KUKA KRL program: ps_603res_c1_orig.src, ps_603res_c1_orig.dat

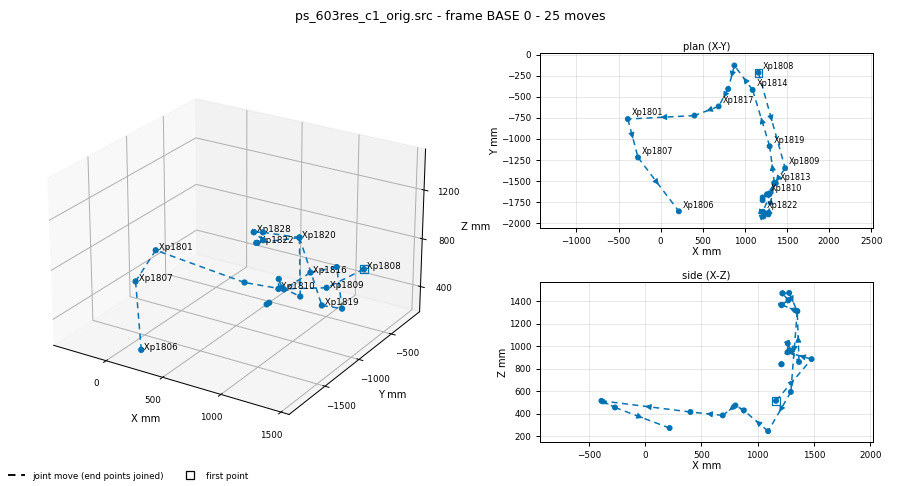
[picture p0: tool path of ps_603res_c1_orig.src in frame BASE 0, 25 of 40 moves have a stored position in this frame; points joined in program order, loops and branches not executed]
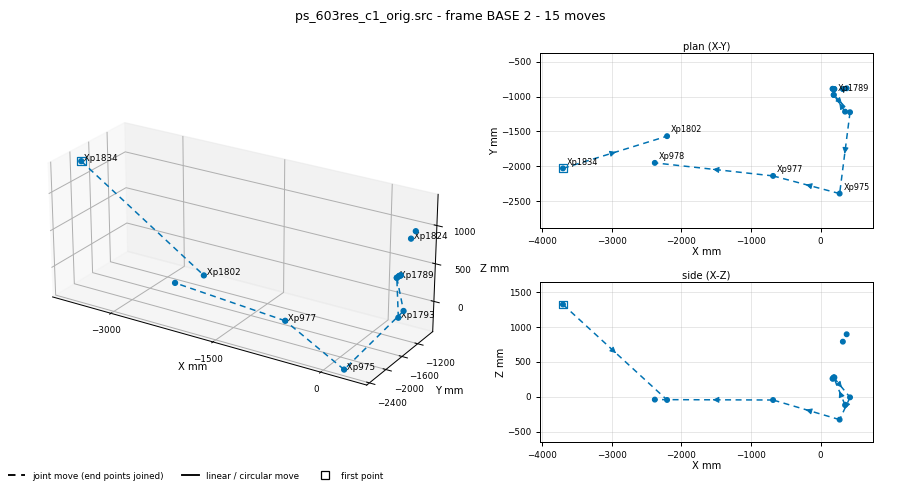
[picture p1: tool path of ps_603res_c1_orig.src in frame BASE 2, 15 of 40 moves have a stored position in this frame; points joined in program order, loops and branches not executed]
--- ps_603res_c1_orig.src ---
&ACCESS RVO
&COMMENT Solda Respot Geo1 C1
DEF ps_603res_c1_orig( )
EXT e_Fraes1 ( )
EXT f_Fraes1 ( )

  ;FOLD INI;%{PE}%V2.2.2,%MKUKATPBASIS,%CINIT,%VCOMMON,%P
  ;FOLD BAS INI;%{PE}%V2.2.2,%MKUKATPBASIS,%CINIT,%VINIT,%P
  INTERRUPT DECL 3 WHEN $STOPMESS==TRUE DO IR_STOPM ( )
  INTERRUPT ON 3
  BAS (#INITMOV,0 )
  ;ENDFOLD
  ;FOLD A20 INI;%{E}%V2.2.2,%MKUKATPA20,%CINIT,%VINIT,%P
  IF ARC20==TRUE THEN
    A20 (ARC_INI)
    INTERRUPT DECL 6 WHEN $CYCFLAG[3]==FALSE DO A20(TECH_STOP2)
  ENDIF
  ;ENDFOLD
  ;FOLD A10 INI;%{E}%V2.2.2,%MKUKATPARC,%CINIT,%VINIT,%P
  IF A10_OPTION==#ACTIVE THEN
    INTERRUPT DECL 4 WHEN $CYCFLAG[2]==FALSE DO A10 (#APPL_ERROR)
    INTERRUPT DECL 7 WHEN A_ARC_SWI==#ACTIVE DO A10 (#ARC_SEAM)
    INTERRUPT DECL 5 WHEN A_FLY_ARC==TRUE DO A10 (#HPU_ARC)
    INTERRUPT  ON 5
    A10_INI ( )
  ENDIF
  ;ENDFOLD
  ;FOLD GRIPPER INI;%{E}%V2.2.2,%MKUKATPGRIPPER,%CINIT,%VINIT,%P
  USER_GRP(0,DUMMY,DUMMY,GDEFAULT)
  ;ENDFOLD
  ;FOLD SPOT INI;%{E}%V.2.2,%MKUKATPSPOT,%CINIT,%VINIT,%P
  USERSPOT(#INIT)
  ;ENDFOLD
  ;FOLD TOUCHSENSE INI;%{E}%V2.2.2,%MKUKATPTS,%CINIT,%VINIT,%P
  IF H70_OPTION THEN
    INTERRUPT DECL 15 WHEN $MEAS_PULSE[TOUCH_I[TOUCH_ACTIVE].IN_NR] DO H70 (6,CD0 )
    INTERRUPT DECL 16 WHEN $ZERO_MOVE DO H70 (7,CD0 )
    INTERRUPT DECL 17 WHEN $TECHPAR_C[FG_TOUCH,8]>0.5 DO H70 (8,CD0)
    H70 (1,CD0 )
  ENDIF
  ;ENDFOLD
  ;FOLD USER INI;%{P}%V2.2.2,%MKUKATPUSER,%CINIT,%VINIT,%P
  ;Make your modifications here
  ;ENDFOLD
  ;ENDFOLD

; Caracterização dos meios de produção:
; Versão Atual:
; 19/07/2013 12:00 Name: P13.060-R3 CHANGES: Solda respot C1
; Accelo

chk_w1_wechs_ok ( )        ;VERIFICAÇÃO DE FERRAMENTA: C1

;FOLD PTP p1834  Vel= 80 % PDAT43 Tool[1]:Gun C1 Base[2]:Accelo;%{PE}%R 4.1.16,%MKUKATPBASIS,%CMOVE,%VPTP,%P 1:PTP, 2:p1834, 3:, 5:80, 7:PDAT43
$BWDSTART = FALSE
PDAT_ACT=PPDAT43
BAS(#PTP_DAT)
FDAT_ACT=Fp1834
BAS(#FRAMES)
BAS(#VEL_PTP,80)
PTP Xp1834
;ENDFOLD
;FOLD PTP p1802  Vel= 80 % PDAT11 Tool[1]:Gun C1 Base[2]:Accelo;%{PE}%R 4.1.16,%MKUKATPBASIS,%CMOVE,%VPTP,%P 1:PTP, 2:p1802, 3:, 5:80, 7:PDAT11
$BWDSTART = FALSE
PDAT_ACT=PPDAT11
BAS(#PTP_DAT)
FDAT_ACT=Fp1802
BAS(#FRAMES)
BAS(#VEL_PTP,80)
PTP Xp1802
;ENDFOLD

;FOLD OUT 838 'Solic. Lib. Soldar Respot GEO 1'  State= TRUE ;%{PE}%R 4.1.16,%MKUKATPBASIS,%COUT,%VOUTX,%P 2:838, 3:'Solic. Lib. Soldar Respot GEO 1', 5:TRUE, 6:
$OUT[838]=TRUE
;ENDFOLD
;FOLD WAIT FOR IN 846 'Aguarda lib. soldar respot Geo1'  State= TRUE ;%{PE}%R 4.1.16,%MKUKATPBASIS,%CWAIT_FOR,%VWAIT_FOR,%P 1:0, 2:846, 3:'Aguarda lib. soldar respot Geo1', 5:TRUE, 6:
WAIT FOR $IN[846]==TRUE
;ENDFOLD
;FOLD OUT 838 'Solic. Lib. Soldar Respot GEO 1'  State= FALSE ;%{PE}%R 4.1.16,%MKUKATPBASIS,%COUT,%VOUTX,%P 2:838, 3:'Solic. Lib. Soldar Respot GEO 1', 5:FALSE, 6:
$OUT[838]=FALSE
;ENDFOLD

;FOLD OUT 851 'Libera  AGV'  State= FALSE ;%{PE}%R 4.1.16,%MKUKATPBASIS,%COUT,%VOUTX,%P 2:851, 3:'Libera  AGV', 5:FALSE, 6:
$OUT[851]=FALSE
;ENDFOLD

;FOLD Kollision.Ueberwachung_1_Ein ;%{PE}%MKUKATPUSER
COLLSTOP( 1, 1 ) ;INTERRUPTUEBERWACHT
;ENDFOLD

;FOLD PTP p1808  Vel= 80 % PDAT17 Tool[1]:Gun C1 Base[0];%{PE}%R 4.1.16,%MKUKATPBASIS,%CMOVE,%VPTP,%P 1:PTP, 2:p1808, 3:, 5:80, 7:PDAT17
$BWDSTART = FALSE
PDAT_ACT=PPDAT17
BAS(#PTP_DAT)
FDAT_ACT=Fp1808
BAS(#FRAMES)
BAS(#VEL_PTP,80)
PTP Xp1808
;ENDFOLD
;FOLD PTP p1809 CONT Vel= 80 % PDAT18 Tool[1]:Gun C1 Base[0];%{PE}%R 4.1.16,%MKUKATPBASIS,%CMOVE,%VPTP,%P 1:PTP, 2:p1809, 3:C_PTP, 5:80, 7:PDAT18
$BWDSTART = FALSE
PDAT_ACT=PPDAT18
BAS(#PTP_DAT)
FDAT_ACT=Fp1809
BAS(#FRAMES)
BAS(#VEL_PTP,80)
PTP Xp1809 C_PTP
;ENDFOLD
;FOLD PTP p1810 CONT Vel= 80 % PDAT19 Tool[1]:Gun C1 Base[0];%{PE}%R 4.1.16,%MKUKATPBASIS,%CMOVE,%VPTP,%P 1:PTP, 2:p1810, 3:C_PTP, 5:80, 7:PDAT19
$BWDSTART = FALSE
PDAT_ACT=PPDAT19
BAS(#PTP_DAT)
FDAT_ACT=Fp1810
BAS(#FRAMES)
BAS(#VEL_PTP,80)
PTP Xp1810 C_PTP
;ENDFOLD

;FOLD PTP SWP_62_0005 PDAT20 SPOT Gun= 1 RETR OPN PgNo1= 36 ACTIVE= 1 Tool[1]:Gun C1 Base[0];%{PE}%R 4.1.12,%MKUKATPSPOT,%CSPOT,%VPTP,%P 1:PTP, 2:SWP_62_0005, 3:, 5:80, 7:PDAT20, 10:1, 12:#FIRST, 14:#OPN, 16:36, 18:1, 20:0, 22:0, 24:1, 25:NORMAL
$BWDSTART = FALSE
PDAT_ACT=PPDAT20
BAS(#PTP_DAT)
FDAT_ACT=FSWP_62_0005
BAS(#FRAMES)
BAS(#VEL_PTP,PPDAT20.VEL)
S_ACT.GUN=1
S_ACT.PAIR=SDEFAULT.PAIR
S_ACT.RETR=#OPN
S_ACT.CLO_TM=1
S_ACT.PGNO1=36
S_ACT.PGNO2=SDEFAULT.PGNO2
S_ACT.PRESS1=SDEFAULT.PRESS1
S_ACT.PRESS2=SDEFAULT.PRESS2
S_READY=FALSE
PTP XSWP_62_0005
USERSPOT(#SPOT, S_ACT)
WAIT FOR S_READY
;ENDFOLD

;FOLD PTP p1812 CONT Vel= 80 % PDAT21 Tool[1]:Gun C1 Base[0];%{PE}%R 4.1.16,%MKUKATPBASIS,%CMOVE,%VPTP,%P 1:PTP, 2:p1812, 3:C_PTP, 5:80, 7:PDAT21
$BWDSTART = FALSE
PDAT_ACT=PPDAT21
BAS(#PTP_DAT)
FDAT_ACT=Fp1812
BAS(#FRAMES)
BAS(#VEL_PTP,80)
PTP Xp1812 C_PTP
;ENDFOLD
;FOLD PTP p1813 CONT Vel= 80 % PDAT22 Tool[1]:Gun C1 Base[0];%{PE}%R 4.1.16,%MKUKATPBASIS,%CMOVE,%VPTP,%P 1:PTP, 2:p1813, 3:C_PTP, 5:80, 7:PDAT22
$BWDSTART = FALSE
PDAT_ACT=PPDAT22
BAS(#PTP_DAT)
FDAT_ACT=Fp1813
BAS(#FRAMES)
BAS(#VEL_PTP,80)
PTP Xp1813 C_PTP
;ENDFOLD
;FOLD PTP p1820  Vel= 80 % PDAT29 Tool[1]:Gun C1 Base[0];%{PE}%R 4.1.16,%MKUKATPBASIS,%CMOVE,%VPTP,%P 1:PTP, 2:p1820, 3:, 5:80, 7:PDAT29
$BWDSTART = FALSE
PDAT_ACT=PPDAT29
BAS(#PTP_DAT)
FDAT_ACT=Fp1820
BAS(#FRAMES)
BAS(#VEL_PTP,80)
PTP Xp1820
;ENDFOLD
;FOLD PTP p1822  Vel= 80 % PDAT31 Tool[1]:Gun C1 Base[0];%{PE}%R 4.1.16,%MKUKATPBASIS,%CMOVE,%VPTP,%P 1:PTP, 2:p1822, 3:, 5:80, 7:PDAT31
$BWDSTART = FALSE
PDAT_ACT=PPDAT31
BAS(#PTP_DAT)
FDAT_ACT=Fp1822
BAS(#FRAMES)
BAS(#VEL_PTP,80)
PTP Xp1822
;ENDFOLD

;FOLD PTP p1824 PDAT33 SPOT Gun= 1 RETR OPN PgNo1= 1 ACTIVE= 1 Tool[1]:Gun C1 Base[2]:Accelo;%{PE}%R 4.1.12,%MKUKATPSPOT,%CSPOT,%VPTP,%P 1:PTP, 2:p1824, 3:, 5:80, 7:PDAT33, 10:1, 12:#FIRST, 14:#OPN, 16:1, 18:1, 20:0, 22:0, 24:1, 25:NORMAL
$BWDSTART = FALSE
PDAT_ACT=PPDAT33
BAS(#PTP_DAT)
FDAT_ACT=Fp1824
BAS(#FRAMES)
BAS(#VEL_PTP,PPDAT33.VEL)
S_ACT.GUN=1
S_ACT.PAIR=SDEFAULT.PAIR
S_ACT.RETR=#OPN
S_ACT.CLO_TM=1
S_ACT.PGNO1=1
S_ACT.PGNO2=SDEFAULT.PGNO2
S_ACT.PRESS1=SDEFAULT.PRESS1
S_ACT.PRESS2=SDEFAULT.PRESS2
S_READY=FALSE
PTP Xp1824
USERSPOT(#SPOT, S_ACT)
WAIT FOR S_READY
;ENDFOLD

;FOLD PTP p1825  Vel= 80 % PDAT34 Tool[1]:Gun C1 Base[0];%{PE}%R 4.1.16,%MKUKATPBASIS,%CMOVE,%VPTP,%P 1:PTP, 2:p1825, 3:, 5:80, 7:PDAT34
$BWDSTART = FALSE
PDAT_ACT=PPDAT34
BAS(#PTP_DAT)
FDAT_ACT=Fp1825
BAS(#FRAMES)
BAS(#VEL_PTP,80)
PTP Xp1825
;ENDFOLD
;FOLD PTP p1826  Vel= 80 % PDAT35 Tool[1]:Gun C1 Base[0];%{PE}%R 4.1.16,%MKUKATPBASIS,%CMOVE,%VPTP,%P 1:PTP, 2:p1826, 3:, 5:80, 7:PDAT35
$BWDSTART = FALSE
PDAT_ACT=PPDAT35
BAS(#PTP_DAT)
FDAT_ACT=Fp1826
BAS(#FRAMES)
BAS(#VEL_PTP,80)
PTP Xp1826
;ENDFOLD
;FOLD PTP p1828  Vel= 80 % PDAT37 Tool[1]:Gun C1 Base[0];%{PE}%R 4.1.16,%MKUKATPBASIS,%CMOVE,%VPTP,%P 1:PTP, 2:p1828, 3:, 5:80, 7:PDAT37
$BWDSTART = FALSE
PDAT_ACT=PPDAT37
BAS(#PTP_DAT)
FDAT_ACT=Fp1828
BAS(#FRAMES)
BAS(#VEL_PTP,80)
PTP Xp1828
;ENDFOLD

;FOLD PTP p1829 PDAT38 SPOT Gun= 1 RETR OPN PgNo1= 1 ACTIVE= 1 Tool[1]:Gun C1 Base[2]:Accelo;%{PE}%R 4.1.12,%MKUKATPSPOT,%CSPOT,%VPTP,%P 1:PTP, 2:p1829, 3:, 5:80, 7:PDAT38, 10:1, 12:#FIRST, 14:#OPN, 16:1, 18:1, 20:0, 22:0, 24:1, 25:NORMAL
$BWDSTART = FALSE
PDAT_ACT=PPDAT38
BAS(#PTP_DAT)
FDAT_ACT=Fp1829
BAS(#FRAMES)
BAS(#VEL_PTP,PPDAT38.VEL)
S_ACT.GUN=1
S_ACT.PAIR=SDEFAULT.PAIR
S_ACT.RETR=#OPN
S_ACT.CLO_TM=1
S_ACT.PGNO1=1
S_ACT.PGNO2=SDEFAULT.PGNO2
S_ACT.PRESS1=SDEFAULT.PRESS1
S_ACT.PRESS2=SDEFAULT.PRESS2
S_READY=FALSE
PTP Xp1829
USERSPOT(#SPOT, S_ACT)
WAIT FOR S_READY
;ENDFOLD

;FOLD PTP p1830  Vel= 80 % PDAT39 Tool[1]:Gun C1 Base[0];%{PE}%R 4.1.16,%MKUKATPBASIS,%CMOVE,%VPTP,%P 1:PTP, 2:p1830, 3:, 5:80, 7:PDAT39
$BWDSTART = FALSE
PDAT_ACT=PPDAT39
BAS(#PTP_DAT)
FDAT_ACT=Fp1830
BAS(#FRAMES)
BAS(#VEL_PTP,80)
PTP Xp1830
;ENDFOLD
;FOLD PTP p1831  Vel= 80 % PDAT40 Tool[1]:Gun C1 Base[0];%{PE}%R 4.1.16,%MKUKATPBASIS,%CMOVE,%VPTP,%P 1:PTP, 2:p1831, 3:, 5:80, 7:PDAT40
$BWDSTART = FALSE
PDAT_ACT=PPDAT40
BAS(#PTP_DAT)
FDAT_ACT=Fp1831
BAS(#FRAMES)
BAS(#VEL_PTP,80)
PTP Xp1831
;ENDFOLD
;FOLD PTP p1832  Vel= 80 % PDAT41 Tool[1]:Gun C1 Base[0];%{PE}%R 4.1.16,%MKUKATPBASIS,%CMOVE,%VPTP,%P 1:PTP, 2:p1832, 3:, 5:80, 7:PDAT41
$BWDSTART = FALSE
PDAT_ACT=PPDAT41
BAS(#PTP_DAT)
FDAT_ACT=Fp1832
BAS(#FRAMES)
BAS(#VEL_PTP,80)
PTP Xp1832
;ENDFOLD
;FOLD PTP p1819  Vel= 80 % PDAT28 Tool[1]:Gun C1 Base[0];%{PE}%R 4.1.16,%MKUKATPBASIS,%CMOVE,%VPTP,%P 1:PTP, 2:p1819, 3:, 5:80, 7:PDAT28
$BWDSTART = FALSE
PDAT_ACT=PPDAT28
BAS(#PTP_DAT)
FDAT_ACT=Fp1819
BAS(#FRAMES)
BAS(#VEL_PTP,80)
PTP Xp1819
;ENDFOLD
;FOLD PTP p1814 CONT Vel= 80 % PDAT23 Tool[1]:Gun C1 Base[0];%{PE}%R 4.1.16,%MKUKATPBASIS,%CMOVE,%VPTP,%P 1:PTP, 2:p1814, 3:C_PTP, 5:80, 7:PDAT23
$BWDSTART = FALSE
PDAT_ACT=PPDAT23
BAS(#PTP_DAT)
FDAT_ACT=Fp1814
BAS(#FRAMES)
BAS(#VEL_PTP,80)
PTP Xp1814 C_PTP
;ENDFOLD
;FOLD PTP p1815 CONT Vel= 80 % PDAT24 Tool[1]:Gun C1 Base[0];%{PE}%R 4.1.16,%MKUKATPBASIS,%CMOVE,%VPTP,%P 1:PTP, 2:p1815, 3:C_PTP, 5:80, 7:PDAT24
$BWDSTART = FALSE
PDAT_ACT=PPDAT24
BAS(#PTP_DAT)
FDAT_ACT=Fp1815
BAS(#FRAMES)
BAS(#VEL_PTP,80)
PTP Xp1815 C_PTP
;ENDFOLD
;FOLD PTP p1816 CONT Vel= 80 % PDAT25 Tool[1]:Gun C1 Base[0];%{PE}%R 4.1.16,%MKUKATPBASIS,%CMOVE,%VPTP,%P 1:PTP, 2:p1816, 3:C_PTP, 5:80, 7:PDAT25
$BWDSTART = FALSE
PDAT_ACT=PPDAT25
BAS(#PTP_DAT)
FDAT_ACT=Fp1816
BAS(#FRAMES)
BAS(#VEL_PTP,80)
PTP Xp1816 C_PTP
;ENDFOLD
;FOLD PTP p1817 CONT Vel= 80 % PDAT26 Tool[1]:Gun C1 Base[0];%{PE}%R 4.1.16,%MKUKATPBASIS,%CMOVE,%VPTP,%P 1:PTP, 2:p1817, 3:C_PTP, 5:80, 7:PDAT26
$BWDSTART = FALSE
PDAT_ACT=PPDAT26
BAS(#PTP_DAT)
FDAT_ACT=Fp1817
BAS(#FRAMES)
BAS(#VEL_PTP,80)
PTP Xp1817 C_PTP
;ENDFOLD
;FOLD PTP p1818 CONT Vel= 80 % PDAT27 Tool[1]:Gun C1 Base[0];%{PE}%R 4.1.16,%MKUKATPBASIS,%CMOVE,%VPTP,%P 1:PTP, 2:p1818, 3:C_PTP, 5:80, 7:PDAT27
$BWDSTART = FALSE
PDAT_ACT=PPDAT27
BAS(#PTP_DAT)
FDAT_ACT=Fp1818
BAS(#FRAMES)
BAS(#VEL_PTP,80)
PTP Xp1818 C_PTP
;ENDFOLD
;FOLD PTP p1801 CONT Vel= 80 % PDAT10 Tool[1]:Gun C1 Base[0];%{PE}%R 4.1.16,%MKUKATPBASIS,%CMOVE,%VPTP,%P 1:PTP, 2:p1801, 3:C_PTP, 5:80, 7:PDAT10
$BWDSTART = FALSE
PDAT_ACT=PPDAT10
BAS(#PTP_DAT)
FDAT_ACT=Fp1801
BAS(#FRAMES)
BAS(#VEL_PTP,80)
PTP Xp1801 C_PTP
;ENDFOLD
;FOLD PTP p1807 CONT Vel= 80 % PDAT16 Tool[1]:Gun C1 Base[0];%{PE}%R 4.1.16,%MKUKATPBASIS,%CMOVE,%VPTP,%P 1:PTP, 2:p1807, 3:C_PTP, 5:80, 7:PDAT16
$BWDSTART = FALSE
PDAT_ACT=PPDAT16
BAS(#PTP_DAT)
FDAT_ACT=Fp1807
BAS(#FRAMES)
BAS(#VEL_PTP,80)
PTP Xp1807 C_PTP
;ENDFOLD
;FOLD PTP p1806  Vel= 80 % PDAT15 Tool[1]:Gun C1 Base[0];%{PE}%R 4.1.16,%MKUKATPBASIS,%CMOVE,%VPTP,%P 1:PTP, 2:p1806, 3:, 5:80, 7:PDAT15
$BWDSTART = FALSE
PDAT_ACT=PPDAT15
BAS(#PTP_DAT)
FDAT_ACT=Fp1806
BAS(#FRAMES)
BAS(#VEL_PTP,80)
PTP Xp1806
;ENDFOLD

;FOLD OUT 838 'Solic. Lib. Soldar Respot GEO 1'  State= TRUE ;%{PE}%R 4.1.16,%MKUKATPBASIS,%COUT,%VOUTX,%P 2:838, 3:'Solic. Lib. Soldar Respot GEO 1', 5:TRUE, 6:
$OUT[838]=TRUE
;ENDFOLD
;FOLD WAIT FOR IN 846 'aguarda lib. soldar respot Geo1'  State= TRUE ;%{PE}%R 4.1.16,%MKUKATPBASIS,%CWAIT_FOR,%VWAIT_FOR,%P 1:0, 2:846, 3:'aguarda lib. soldar respot Geo1', 5:TRUE, 6:
WAIT FOR $IN[846]==TRUE
;ENDFOLD
;FOLD OUT 838 'Solic. Lib. Soldar Respot GEO 1'  State= FALSE ;%{PE}%R 4.1.16,%MKUKATPBASIS,%COUT,%VOUTX,%P 2:838, 3:'Solic. Lib. Soldar Respot GEO 1', 5:FALSE, 6:
$OUT[838]=FALSE
;ENDFOLD

;FOLD PTP p1793 CONT Vel= 65 % PDAT7 Tool[1]:Gun C1 Base[2]:Accelo;%{PE}%R 4.1.16,%MKUKATPBASIS,%CMOVE,%VPTP,%P 1:PTP, 2:p1793, 3:C_PTP, 5:65, 7:PDAT7
$BWDSTART = FALSE
PDAT_ACT=PPDAT7
BAS(#PTP_DAT)
FDAT_ACT=Fp1793
BAS(#FRAMES)
BAS(#VEL_PTP,65)
PTP Xp1793 C_PTP
;ENDFOLD
;FOLD PTP p1789  Vel= 75 % PDAT3 Tool[1]:Gun C1 Base[2]:Accelo;%{PE}%R 4.1.16,%MKUKATPBASIS,%CMOVE,%VPTP,%P 1:PTP, 2:p1789, 3:, 5:75, 7:PDAT3
$BWDSTART = FALSE
PDAT_ACT=PPDAT3
BAS(#PTP_DAT)
FDAT_ACT=Fp1789
BAS(#FRAMES)
BAS(#VEL_PTP,75)
PTP Xp1789
;ENDFOLD

;FOLD OUT 839 'Soldando'  State= TRUE ;%{PE}%R 4.1.16,%MKUKATPBASIS,%COUT,%VOUTX,%P 2:839, 3:'Soldando', 5:TRUE, 6:
$OUT[839]=TRUE
;ENDFOLD
;FOLD OUT 848 'Area de Solda'  State= FALSE ;%{PE}%R 4.1.16,%MKUKATPBASIS,%COUT,%VOUTX,%P 2:848, 3:'Area de Solda', 5:FALSE, 6:
$OUT[848]=FALSE
;ENDFOLD

;FOLD LIN p1794 CONT Vel= 2 m/s CPDAT14 Tool[1]:Gun C1 Base[2]:Accelo;%{PE}%R 4.1.16,%MKUKATPBASIS,%CMOVE,%VLIN,%P 1:LIN, 2:p1794, 3:C_DIS, 5:2, 7:CPDAT14
$BWDSTART = FALSE
LDAT_ACT=LCPDAT14
BAS(#CP_DAT)
FDAT_ACT=Fp1794
BAS(#FRAMES)
BAS(#VEL_CP,2)
LIN Xp1794 C_DIS
;ENDFOLD

;FOLD ; SWP_60_0213;%{PE}%R 4.1.16,%MKUKATPBASIS,%CCOMMENT,%VNORMAL,%P 2:SWP_60_0213
;ENDFOLD
;FOLD LIN swp_60_0213 CPDAT16 SPOT Gun= 1 RETR OPN PgNo1= 14 ACTIVE= 1 Tool[1]:Gun C1 Base[0];%{PE}%R 4.1.12,%MKUKATPSPOT,%CSPOT,%VLIN,%P 1:LIN, 2:swp_60_0213, 3:, 5:2, 7:CPDAT16, 10:1, 12:#FIRST, 14:#OPN, 16:14, 18:1, 20:0, 22:0, 24:1, 25:NORMAL
$BWDSTART = FALSE
LDAT_ACT=LCPDAT16
BAS(#CP_DAT)
FDAT_ACT=Fswp_60_0213
BAS(#FRAMES)
BAS(#VEL_CP,LCPDAT16.VEL)
S_ACT.GUN=1
S_ACT.PAIR=SDEFAULT.PAIR
S_ACT.RETR=#OPN
S_ACT.CLO_TM=1
S_ACT.PGNO1=14
S_ACT.PGNO2=SDEFAULT.PGNO2
S_ACT.PRESS1=SDEFAULT.PRESS1
S_ACT.PRESS2=SDEFAULT.PRESS2
S_READY=FALSE
LIN Xswp_60_0213
USERSPOT(#SPOT, S_ACT)
WAIT FOR S_READY
;ENDFOLD

;FOLD LIN p1795 CONT Vel= 2 m/s CPDAT15 Tool[1]:Gun C1 Base[2]:Accelo;%{PE}%R 4.1.16,%MKUKATPBASIS,%CMOVE,%VLIN,%P 1:LIN, 2:p1795, 3:C_DIS, 5:2, 7:CPDAT15
$BWDSTART = FALSE
LDAT_ACT=LCPDAT15
BAS(#CP_DAT)
FDAT_ACT=Fp1795
BAS(#FRAMES)
BAS(#VEL_CP,2)
LIN Xp1795 C_DIS
;ENDFOLD

;FOLD ; SWP_60_0215;%{PE}%R 4.1.16,%MKUKATPBASIS,%CCOMMENT,%VNORMAL,%P 2:SWP_60_0215
;ENDFOLD
;FOLD LIN swp_60_0215 CPDAT19 SPOT Gun= 1 RETR OPN PgNo1= 15 ACTIVE= 1 Tool[1]:Gun C1 Base[0];%{PE}%R 4.1.12,%MKUKATPSPOT,%CSPOT,%VLIN,%P 1:LIN, 2:swp_60_0215, 3:, 5:2, 7:CPDAT19, 10:1, 12:#FIRST, 14:#OPN, 16:15, 18:1, 20:0, 22:0, 24:1, 25:NORMAL
$BWDSTART = FALSE
LDAT_ACT=LCPDAT19
BAS(#CP_DAT)
FDAT_ACT=Fswp_60_0215
BAS(#FRAMES)
BAS(#VEL_CP,LCPDAT19.VEL)
S_ACT.GUN=1
S_ACT.PAIR=SDEFAULT.PAIR
S_ACT.RETR=#OPN
S_ACT.CLO_TM=1
S_ACT.PGNO1=15
S_ACT.PGNO2=SDEFAULT.PGNO2
S_ACT.PRESS1=SDEFAULT.PRESS1
S_ACT.PRESS2=SDEFAULT.PRESS2
S_READY=FALSE
LIN Xswp_60_0215
USERSPOT(#SPOT, S_ACT)
WAIT FOR S_READY
;ENDFOLD

;FOLD LIN p1797 CONT Vel= 2 m/s CPDAT18 Tool[1]:Gun C1 Base[2]:Accelo;%{PE}%R 4.1.16,%MKUKATPBASIS,%CMOVE,%VLIN,%P 1:LIN, 2:p1797, 3:C_DIS, 5:2, 7:CPDAT18
$BWDSTART = FALSE
LDAT_ACT=LCPDAT18
BAS(#CP_DAT)
FDAT_ACT=Fp1797
BAS(#FRAMES)
BAS(#VEL_CP,2)
LIN Xp1797 C_DIS
;ENDFOLD

;FOLD OUT 839 'Soldando'  State= FALSE ;%{PE}%R 4.1.16,%MKUKATPBASIS,%COUT,%VOUTX,%P 2:839, 3:'Soldando', 5:FALSE, 6:
$OUT[839]=FALSE
;ENDFOLD
;FOLD OUT 848 'Area de Solda'  State= TRUE ;%{PE}%R 4.1.16,%MKUKATPBASIS,%COUT,%VOUTX,%P 2:848, 3:'Area de Solda', 5:TRUE, 6:
$OUT[848]=TRUE
;ENDFOLD

;FOLD LIN p1798 CONT Vel= 2 m/s CPDAT20 Tool[1]:Gun C1 Base[2]:Accelo;%{PE}%R 4.1.16,%MKUKATPBASIS,%CMOVE,%VLIN,%P 1:LIN, 2:p1798, 3:C_DIS, 5:2, 7:CPDAT20
$BWDSTART = FALSE
LDAT_ACT=LCPDAT20
BAS(#CP_DAT)
FDAT_ACT=Fp1798
BAS(#FRAMES)
BAS(#VEL_CP,2)
LIN Xp1798 C_DIS
;ENDFOLD

;FOLD PTP p973 CONT Vel= 80 % P_OLP11 Tool[1]:Gun C1 Base[2]:Accelo;%{PE}%R 4.1.16,%MKUKATPBASIS,%CMOVE,%VPTP,%P 1:PTP, 2:p973, 3:C_PTP, 5:80, 7:P_OLP11
$BWDSTART = FALSE
PDAT_ACT=PP_OLP11
BAS(#PTP_DAT)
FDAT_ACT=Fp973
BAS(#FRAMES)
BAS(#VEL_PTP,80)
PTP Xp973 C_PTP
;ENDFOLD
;FOLD PTP p974 CONT Vel= 80 % P_OLP12 Tool[1]:Gun C1 Base[2]:Accelo;%{PE}%R 4.1.16,%MKUKATPBASIS,%CMOVE,%VPTP,%P 1:PTP, 2:p974, 3:C_PTP, 5:80, 7:P_OLP12
$BWDSTART = FALSE
PDAT_ACT=PP_OLP12
BAS(#PTP_DAT)
FDAT_ACT=Fp974
BAS(#FRAMES)
BAS(#VEL_PTP,80)
PTP Xp974 C_PTP
;ENDFOLD
;FOLD PTP p975 CONT Vel= 80 % P_OLP13 Tool[1]:Gun C1 Base[2]:Accelo;%{PE}%R 4.1.16,%MKUKATPBASIS,%CMOVE,%VPTP,%P 1:PTP, 2:p975, 3:C_PTP, 5:80, 7:P_OLP13
$BWDSTART = FALSE
PDAT_ACT=PP_OLP13
BAS(#PTP_DAT)
FDAT_ACT=Fp975
BAS(#FRAMES)
BAS(#VEL_PTP,80)
PTP Xp975 C_PTP
;ENDFOLD
;FOLD PTP p977  Vel= 80 % P_OLP15 Tool[1]:Gun C1 Base[2]:Accelo;%{PE}%R 4.1.16,%MKUKATPBASIS,%CMOVE,%VPTP,%P 1:PTP, 2:p977, 3:, 5:80, 7:P_OLP15
$BWDSTART = FALSE
PDAT_ACT=PP_OLP15
BAS(#PTP_DAT)
FDAT_ACT=Fp977
BAS(#FRAMES)
BAS(#VEL_PTP,80)
PTP Xp977
;ENDFOLD

;FOLD ; END INTERLOCK COM R1;%{PE}%R 4.1.16,%MKUKATPBASIS,%CCOMMENT,%VNORMAL,%P 2:END INTERLOCK COM R1
;ENDFOLD
;FOLD Kollision.Ueberwachung_1_Aus ;%{PE}%MKUKATPUSER
COLLSTOP( 1, 2 )
;ENDFOLD

;FOLD PULSE 846 'R3 solda respot Geo 1 concluida'  State= TRUE   Time= 3 sec;%{PE}%R 4.1.16,%MKUKATPBASIS,%COUT,%VPULSE,%P 2:846, 3:'R3 solda respot Geo 1 concluida', 5:TRUE, 6:, 8:3
PULSE($OUT[846], TRUE,3)
;ENDFOLD

;FOLD PTP p978 CONT Vel= 100 % P_OLP16 Tool[1]:Gun C1 Base[2]:Accelo;%{PE}%R 4.1.16,%MKUKATPBASIS,%CMOVE,%VPTP,%P 1:PTP, 2:p978, 3:C_PTP, 5:100, 7:P_OLP16
$BWDSTART = FALSE
PDAT_ACT=PP_OLP16
BAS(#PTP_DAT)
FDAT_ACT=Fp978
BAS(#FRAMES)
BAS(#VEL_PTP,100)
PTP Xp978 C_PTP
;ENDFOLD

IF ((GHOST() OR $IN[821])) THEN
;FOLD OUT 176 'Proteção da pinca 2 fechar'  State= FALSE ;%{PE}%R 4.1.16,%MKUKATPBASIS,%COUT,%VOUTX,%P 2:176, 3:'Proteção da pinca 2 fechar', 5:FALSE, 6:
$OUT[176]=FALSE
;ENDFOLD
;FOLD OUT 175 'Proteção da pinca 2 abrir'  State= TRUE ;%{PE}%R 4.1.16,%MKUKATPBASIS,%COUT,%VOUTX,%P 2:175, 3:'Proteção da pinca 2 abrir', 5:TRUE, 6:
$OUT[175]=TRUE
;ENDFOLD
ENDIF

END

--- ps_603res_c1_orig.dat ---
&ACCESS RVO
&COMMENT Solda Respot Geo1 C1
DEFDAT ps_603res_c1_orig
;FOLD EXTERNAL DECLARATIONS;%{PE}%V2.2.2,%MKUKATPBASIS,%CEXT,%VCOMMON,%P
;FOLD BAS EXT;%{PE}%V2.2.2,%MKUKATPBASIS,%CEXT,%VEXT,%P
EXT  BAS (BAS_COMMAND  :IN,REAL  :IN )
DECL INT SUCCESS
;ENDFOLD
;FOLD A10 EXT;%{E}%V2.2.2,%MKUKATPARC,%CEXT,%VEXT,%P
EXT  A10 (A_CMD_T  :IN,A_STRT_T  :IN,A_WELD_T  :IN,A_END_T  :IN,INT  :IN )
;ENDFOLD
;FOLD A20 EXT;%{E}%V2.2.2,%MKUKATPA20,%CEXT,%VEXT,%P
EXT  A20 (INT  :IN,WELD_ST  :IN,WELD_FI  :IN,INT  :IN )
;ENDFOLD
;FOLD GRIPPER EXT;%{E}%V2.2.2,%MKUKATPGRIPPER,%CEXT,%VEXT,%P
EXT  H50 (INT  :IN,INT  :IN,INT  :IN,GRP_TYP  :IN )
;ENDFOLD
;FOLD SPOT EXT;%{E}%V2.2.2,%MKUKATPSPOT,%CEXT,%VEXT,%P
EXT  USERSPOT (S_COMMAND  :IN,SPOT_TYPE  :IN )
;ENDFOLD
;FOLD TOUCHSENSE EXT;%{E}%V2.2.2,%MKUKATPTS,%CEXT,%VEXT,%P
EXT  H70 (INT  :IN,SRCH_TYP_2  :OUT,E6POS  :IN,SRCH_TYP_3  :IN,SRCH_TYP_2  :IN,SRCH_TYP_2  :IN,SRCH_TYP_2  :IN,SRCH_TYP_2  :IN,SRCH_TYP_2  :IN,INT  :IN )
;ENDFOLD
;FOLD USER EXT;%{}%V2.2.2,%MKUKATPUSER,%CEXT,%VEXT,%P
;Make here your modifications
;ENDFOLD
;ENDFOLD

;# ============ START PATH : swp_p13060r3_ltc_resp1_c1 =============
DECL FDAT Fp963={TOOL_NO 1,BASE_NO 2,IPO_FRAME #BASE}
DECL PDAT PP_OLP1={VEL 100.0,ACC 100.0,APO_DIST 0.0}
DECL E6POS Xp963={x -3572.9751,y -2107.74902,z 1272.901,a 86.0327988,b 14.4777002,c 74.495903,s 2,t 3}
DECL FDAT Fp964={TOOL_NO 1,BASE_NO 2,IPO_FRAME #BASE}
DECL PDAT PP_OLP2={VEL 100.0,ACC 85.0,APO_DIST 60.0}
DECL E6POS Xp964={x -1796.38599,y -2237.50098,z 3255.19995,a -90.0,b 0.0,c 170.0,s 6,t 51}
DECL FDAT Fp965={TOOL_NO 1,BASE_NO 2,IPO_FRAME #BASE}
DECL PDAT PP_OLP3={VEL 100.0,ACC 85.0,APO_DIST 15.0}
DECL E6POS Xp965={x -1013.56299,y -2243.53296,z 3255.19995,a 70.0,b 0.0,c 170.0,s 6,t 50}
DECL FDAT Fp966={TOOL_NO 1,BASE_NO 2,IPO_FRAME #BASE}
DECL PDAT PP_OLP4={VEL 100.0,ACC 85.0,APO_DIST 20.0}
DECL E6POS Xp966={x -134.343201,y -2313.625,z -64.5488205,a 1.681077,b -1.44535995,c 0.678022921,s 2,t 10,e1 0.0,e2 0.0,e3 0.0,e4 0.0,e5 0.0,e6 0.0}
DECL FDAT Fp967={TOOL_NO 1,BASE_NO 2,IPO_FRAME #BASE}
DECL PDAT PP_OLP5={VEL 100.0,ACC 100.0,APO_DIST 100.0}
DECL E6POS Xp967={x 199.132004,y -934.976013,z 255.951996,a 31.1662006,b 48.9373016,c 116.802299,s 6,t 50}
DECL FDAT Fp968={TOOL_NO 1,BASE_NO 2,IPO_FRAME #BASE}
DECL PDAT PP_OLP6={VEL 100.0,ACC 85.0,APO_DIST 10.0}
DECL E6POS Xp968={x 318.066895,y -1890.32605,z -296.505615,a 6.09352779,b -3.63016009,c 11.6354103,s 2,t 10,e1 0.0,e2 0.0,e3 0.0,e4 0.0,e5 0.0,e6 0.0}
DECL FDAT Fp969={TOOL_NO 1,BASE_NO 2,IPO_FRAME #BASE}
DECL PDAT PP_OLP7={VEL 100.0,ACC 85.0,APO_DIST 5.0}
DECL E6POS Xp969={x 197.508408,y -888.166077,z 282.583313,a 2.79331207,b 35.6193008,c 91.0491791,s 6,t 50,e1 0.0,e2 0.0,e3 0.0,e4 0.0,e5 0.0,e6 0.0}
DECL FDAT Fp970={TOOL_NO 1,BASE_NO 2,IPO_FRAME #BASE}
DECL PDAT PP_OLP8={VEL 100.0,ACC 100.0,APO_DIST 100.0}
DECL E6POS Xp970={x 191.053497,y -889.268982,z 200.622604,a 2.60313106,b 52.9382095,c 92.072197,s 6,t 50,e1 0.0,e2 0.0,e3 0.0,e4 0.0,e5 0.0,e6 0.0}
DECL FDAT Fp971={TOOL_NO 1,BASE_NO 2,IPO_FRAME #BASE}
DECL PDAT PP_OLP9={VEL 100.0,ACC 100.0,APO_DIST 100.0}
DECL E6POS Xp971={x 193.593796,y -886.93158,z 200.001999,a 2.60292602,b 52.9385605,c 92.071907,s 6,t 50,e1 0.0,e2 0.0,e3 0.0,e4 0.0,e5 0.0,e6 0.0}
DECL FDAT Fp972={TOOL_NO 1,BASE_NO 2,IPO_FRAME #BASE}
DECL PDAT PP_OLP10={VEL 100.0,ACC 100.0,APO_DIST 100.0}
DECL E6POS Xp972={x 190.962006,y -887.40802,z 255.615005,a 15.6997004,b 59.0479012,c 103.552902,s 6,t 50}
DECL FDAT Fp973={TOOL_NO 1,BASE_NO 2,IPO_FRAME #BASE}
DECL PDAT PP_OLP11={VEL 100.0,ACC 85.0,APO_DIST 15.0}
DECL E6POS Xp973={x 188.3909,y -976.163513,z 275.360504,a 6.09893894,b 13.9292002,c 94.6382599,s 2,t 10,e1 0.0,e2 0.0,e3 0.0,e4 0.0,e5 0.0,e6 0.0}
DECL FDAT Fp974={TOOL_NO 1,BASE_NO 2,IPO_FRAME #BASE}
DECL PDAT PP_OLP12={VEL 100.0,ACC 85.0,APO_DIST 5.0}
DECL E6POS Xp974={x 422.566498,y -1224.58105,z -8.89597225,a 3.03044891,b -9.06613731,c 48.4070282,s 2,t 10,e1 0.0,e2 0.0,e3 0.0,e4 0.0,e5 0.0,e6 0.0}
DECL FDAT Fp975={TOOL_NO 1,BASE_NO 2,IPO_FRAME #BASE}
DECL PDAT PP_OLP13={VEL 100.0,ACC 85.0,APO_DIST 50.0}
DECL E6POS Xp975={x 273.068604,y -2393.427,z -329.290314,a 5.52923822,b -0.604498804,c -3.24042201,s 2,t 2,e1 0.0,e2 0.0,e3 0.0,e4 0.0,e5 0.0,e6 0.0}
DECL FDAT Fp976={TOOL_NO 1,BASE_NO 2,IPO_FRAME #BASE}
DECL PDAT PP_OLP14={VEL 100.0,ACC 85.0,APO_DIST 30.0}
DECL E6POS Xp976={x -775.734009,y -2495.47412,z -42.9263802,a -127.6604,b 0.485267699,c 4.46799612,s 2,t 2,e1 0.0,e2 0.0,e3 0.0,e4 0.0,e5 0.0,e6 0.0}
DECL FDAT Fp977={TOOL_NO 1,BASE_NO 2,IPO_FRAME #BASE}
DECL PDAT PP_OLP15={VEL 100.0,ACC 85.0,APO_DIST 50.0}
DECL E6POS Xp977={x -683.155823,y -2139.47607,z -47.2864304,a -102.873703,b 0.473506987,c 4.17351484,s 2,t 2,e1 0.0,e2 0.0,e3 0.0,e4 0.0,e5 0.0,e6 0.0}
DECL FDAT Fp978={TOOL_NO 1,BASE_NO 2,IPO_FRAME #BASE}
DECL PDAT PP_OLP16={VEL 100.0,ACC 85.0,APO_DIST 50.0}
DECL E6POS Xp978={x -2382.18701,y -1952.177,z -41.404789,a 68.9136429,b 1.83542502,c 4.31668186,s 2,t 3,e1 0.0,e2 0.0,e3 0.0,e4 0.0,e5 0.0,e6 0.0}
DECL FDAT Fp979={TOOL_NO 1,BASE_NO 2,IPO_FRAME #BASE}
DECL PDAT PP_OLP17={VEL 100.0,ACC 100.0,APO_DIST 100.0}
DECL E6POS Xp979={x -3572.97607,y -2107.75098,z 1272.90002,a 86.0328598,b 14.4777098,c 74.4958572,s 2,t 3,e1 0.0,e2 0.0,e3 0.0,e4 0.0,e5 0.0,e6 0.0}
DECL FDAT Fp980={TOOL_NO 1,BASE_NO 2,IPO_FRAME #BASE}
DECL PDAT PP_OLP18={VEL 100.0,ACC 100.0,APO_DIST 100.0}
DECL E6POS Xp980={x 188.917999,y -888.057983,z 259.154999,a 23.0310001,b 57.8978004,c 109.804703,s 6,t 50}
DECL FDAT Fp981={TOOL_NO 1,BASE_NO 2,IPO_FRAME #BASE}
DECL PDAT PP_OLP19={VEL 100.0,ACC 100.0,APO_DIST 100.0}
DECL E6POS Xp981={x 186.901993,y -888.991028,z 262.647003,a 29.8339005,b 56.3540993,c 115.520699,s 6,t 50}
DECL FDAT Fp982={TOOL_NO 1,BASE_NO 2,IPO_FRAME #BASE}
DECL PDAT PP_OLP20={VEL 100.0,ACC 100.0,APO_DIST 100.0}
DECL E6POS Xp982={x 184.923004,y -890.203979,z 266.074005,a 36.0523987,b 54.4687004,c 120.642502,s 6,t 50}
DECL FDAT Fp983={TOOL_NO 1,BASE_NO 2,IPO_FRAME #BASE}
DECL PDAT PP_OLP21={VEL 100.0,ACC 100.0,APO_DIST 100.0}
DECL E6POS Xp983={x 191.352005,y -892.219971,z 269.428986,a 31.1662006,b 48.9373016,c 116.802299,s 6,t 50}
DECL FDAT Fp984={TOOL_NO 1,BASE_NO 2,IPO_FRAME #BASE}
DECL PDAT PP_OLP22={VEL 100.0,ACC 100.0,APO_DIST 100.0}
DECL E6POS Xp984={x 199.132004,y -934.976013,z 255.951996,a 31.1662006,b 48.9373016,c 116.802299,s 6,t 50}
DECL FDAT Fp985={TOOL_NO 1,BASE_NO 2,IPO_FRAME #BASE}
DECL PDAT PP_OLP23={VEL 100.0,ACC 100.0,APO_DIST 100.0}
DECL E6POS Xp985={x 1034.27002,y -2191.90698,z 1544.59399,a -14.7585001,b 39.6645012,c 130.466705,s 6,t 50}
DECL FDAT Fp986={TOOL_NO 1,BASE_NO 2,IPO_FRAME #BASE}
DECL PDAT PP_OLP24={VEL 100.0,ACC 100.0,APO_DIST 100.0}
DECL E6POS Xp986={x -1013.56299,y -2243.53296,z 3255.19995,a 70.0,b 0.0,c 170.0,s 6,t 50}
DECL FDAT Fp987={TOOL_NO 1,BASE_NO 2,IPO_FRAME #BASE}
DECL PDAT PP_OLP25={VEL 100.0,ACC 100.0,APO_DIST 100.0}
DECL E6POS Xp987={x -1796.38599,y -2237.50098,z 3255.19995,a -90.0,b 0.0,c 170.0,s 6,t 51}
DECL FDAT Fp988={TOOL_NO 1,BASE_NO 2,IPO_FRAME #BASE}
DECL PDAT PP_OLP26={VEL 100.0,ACC 100.0,APO_DIST 0.0}
DECL E6POS Xp988={x -3572.9751,y -2107.74902,z 1272.901,a 86.0327988,b 14.4777002,c 74.495903,s 2,t 3}
DECL SPOT_SUGG_T LAST_SPOT={GUN[] "1                       ",RETR_CMD[] "#OPN                    ",CHOISE[] "#FIRST                  ",CLO_TM[] "1                       ",PGNO1[] "1                       ",PRESS1[] "0                       ",PGNO2[] "1                       ",PRESS2[] "0                       ",SPOT_PARAMS[] "NORMAL                  "}
DECL BASIS_SUGG_T LAST_BASIS={POINT1[] "p1834                   ",POINT2[] "p1834                   ",CP_PARAMS[] "CPDAT20                 ",PTP_PARAMS[] "PDAT43                  ",CONT[] "                        ",CP_VEL[] "2                       ",PTP_VEL[] "80                      "}
DECL E6POS XPS230R01010002={x 1215.79004,y -1725.61401,z 831.992188,a -84.9458389,b 56.91996,c 94.0693436,s 6,t 50,e1 0.0,e2 0.0,e3 0.0,e4 0.0,e5 0.0,e6 0.0}
DECL FDAT FPS230R01010002={TOOL_NO 1,BASE_NO 0,IPO_FRAME #BASE}
DECL PDAT PPDAT1={VEL 60.0,ACC 85.0,APO_DIST 100.0}
DECL E6POS XPS230R01010003={x 1213.63501,y -1696.11401,z 831.111572,a 81.2733688,b 71.3885574,c -99.7629166,s 6,t 50,e1 0.0,e2 0.0,e3 0.0,e4 0.0,e5 0.0,e6 0.0}
DECL FDAT FPS230R01010003={TOOL_NO 1,BASE_NO 0,IPO_FRAME #BASE}
DECL PDAT PPDAT2={VEL 75.0,ACC 85.0,APO_DIST 100.0}
DECL E6POS Xswp_60_0213={x 1210.52905,y -1726.81201,z 839.314514,a -86.5838928,b 67.200882,c 90.8106995,s 2,t 10,e1 0.0,e2 0.0,e3 0.0,e4 0.0,e5 0.0,e6 0.0}
DECL FDAT Fswp_60_0213={TOOL_NO 1,BASE_NO 0,IPO_FRAME #BASE}
DECL E6POS Xswp_60_0215={x 1211.33203,y -1693.92896,z 839.330078,a 87.0061569,b 63.7585793,c -95.0266418,s 2,t 10,e1 0.0,e2 0.0,e3 0.0,e4 0.0,e5 0.0,e6 0.0}
DECL FDAT Fswp_60_0215={TOOL_NO 1,BASE_NO 0,IPO_FRAME #BASE}
DECL E6POS XP1789={x 188.3909,y -976.163513,z 275.360504,a 6.09893894,b 13.9292002,c 94.6382599,s 2,t 10,e1 0.0,e2 0.0,e3 0.0,e4 0.0,e5 0.0,e6 0.0}
DECL FDAT Fp1789={TOOL_NO 1,BASE_NO 2,IPO_FRAME #BASE}
DECL PDAT PPDAT3={VEL 100.0,ACC 85.0,APO_DIST 2.0}
DECL E6POS XP1790={x -775.734009,y -2495.47412,z -42.9263802,a -127.6604,b 0.485267699,c 4.46799612,s 2,t 2,e1 0.0,e2 0.0,e3 0.0,e4 0.0,e5 0.0,e6 0.0}
DECL FDAT Fp1790={TOOL_NO 1,BASE_NO 2,IPO_FRAME #BASE}
DECL PDAT PPDAT4={VEL 100.0,ACC 85.0,APO_DIST 20.0}
DECL E6POS XP1791={x -654.825928,y -2487.59912,z 254.140503,a 62.0100594,b 0.687150598,c -14.3720198,s 6,t 18,e1 0.0,e2 0.0,e3 0.0,e4 0.0,e5 0.0,e6 0.0}
DECL FDAT Fp1791={TOOL_NO 1,BASE_NO 2,IPO_FRAME #BASE}
DECL PDAT PPDAT5={VEL 100.0,ACC 85.0,APO_DIST 20.0}
DECL E6POS XP1792={x -2382.18701,y -1952.177,z -41.404789,a 68.9136429,b 1.83542502,c 4.31668186,s 2,t 3,e1 0.0,e2 0.0,e3 0.0,e4 0.0,e5 0.0,e6 0.0}
DECL FDAT Fp1792={TOOL_NO 1,BASE_NO 2,IPO_FRAME #BASE}
DECL PDAT PPDAT6={VEL 100.0,ACC 85.0,APO_DIST 20.0}
DECL E6POS XP1793={x 351.221191,y -1216.44104,z -120.306999,a 2.85688496,b -3.72620606,c 49.4005203,s 2,t 10,e1 0.0,e2 0.0,e3 0.0,e4 0.0,e5 0.0,e6 0.0}
DECL FDAT Fp1793={TOOL_NO 1,BASE_NO 2,IPO_FRAME #BASE}
DECL PDAT PPDAT7={VEL 100.0,ACC 85.0,APO_DIST 20.0}
DECL E6POS XP1794={x 197.647095,y -891.550476,z 275.967285,a 12.8456602,b 32.3834114,c 97.2856064,s 2,t 10,e1 0.0,e2 0.0,e3 0.0,e4 0.0,e5 0.0,e6 0.0}
DECL FDAT Fp1794={TOOL_NO 1,BASE_NO 2,IPO_FRAME #BASE}
DECL LDAT LCPDAT14={VEL 2.0,ACC 85.0,APO_DIST 5.0,APO_FAC 50.0}
DECL E6POS XP1795={x 173.303894,y -888.536377,z 260.226501,a 41.7541695,b 88.9594727,c 129.317505,s 2,t 10,e1 0.0,e2 0.0,e3 0.0,e4 0.0,e5 0.0,e6 0.0}
DECL FDAT Fp1795={TOOL_NO 1,BASE_NO 2,IPO_FRAME #BASE}
DECL LDAT LCPDAT15={VEL 2.0,ACC 85.0,APO_DIST 5.0,APO_FAC 50.0}
DECL LDAT LCPDAT16={VEL 2.0,ACC 100.0,APO_DIST 100.0,APO_FAC 50.0}
DECL E6POS XP1796={x 154.257401,y -887.912903,z 260.321899,a 178.384201,b 63.5158081,c -93.5807495,s 2,t 10,e1 0.0,e2 0.0,e3 0.0,e4 0.0,e5 0.0,e6 0.0}
DECL FDAT Fp1796={TOOL_NO 1,BASE_NO 2,IPO_FRAME #BASE}
DECL LDAT LCPDAT17={VEL 2.0,ACC 85.0,APO_DIST 5.0,APO_FAC 50.0}
DECL E6POS XP1797={x 173.303406,y -888.314514,z 260.221191,a 41.73423,b 88.9592667,c 129.297501,s 2,t 10,e1 0.0,e2 0.0,e3 0.0,e4 0.0,e5 0.0,e6 0.0}
DECL FDAT Fp1797={TOOL_NO 1,BASE_NO 2,IPO_FRAME #BASE}
DECL LDAT LCPDAT18={VEL 2.0,ACC 85.0,APO_DIST 5.0,APO_FAC 50.0}
DECL LDAT LCPDAT19={VEL 2.0,ACC 100.0,APO_DIST 100.0,APO_FAC 50.0}
DECL E6POS XP1798={x 194.419098,y -891.02478,z 276.474304,a 12.8262901,b 32.2703896,c 97.2526932,s 2,t 10,e1 0.0,e2 0.0,e3 0.0,e4 0.0,e5 0.0,e6 0.0}
DECL FDAT Fp1798={TOOL_NO 1,BASE_NO 2,IPO_FRAME #BASE}
DECL LDAT LCPDAT20={VEL 2.0,ACC 85.0,APO_DIST 5.0,APO_FAC 50.0}
DECL E6POS XP1799={x 273.065491,y -2393.43311,z -329.303894,a 5.53120518,b -0.60386312,c -3.24093199,s 2,t 2,e1 0.0,e2 0.0,e3 0.0,e4 0.0,e5 0.0,e6 0.0}
DECL FDAT Fp1799={TOOL_NO 1,BASE_NO 2,IPO_FRAME #BASE}
DECL PDAT PPDAT8={VEL 100.0,ACC 85.0,APO_DIST 50.0}
DECL E6POS XP1800={x -320.146515,y -2374.72998,z -105.423798,a -2.6406281,b -0.574272275,c 0.858662724,s 2,t 10,e1 0.0,e2 0.0,e3 0.0,e4 0.0,e5 0.0,e6 0.0}
DECL FDAT Fp1800={TOOL_NO 1,BASE_NO 2,IPO_FRAME #BASE}
DECL PDAT PPDAT9={VEL 100.0,ACC 85.0,APO_DIST 10.0}
DECL E6POS XP1801={x -389.750885,y -763.100281,z 514.022827,a 142.2547,b 1.1494,c 4.29426622,s 2,t 2,e1 0.0,e2 0.0,e3 0.0,e4 0.0,e5 0.0,e6 0.0}
DECL FDAT Fp1801={TOOL_NO 1,BASE_NO 0,IPO_FRAME #BASE}
DECL PDAT PPDAT10={VEL 100.0,ACC 85.0,APO_DIST 10.0}
DECL E6POS XP1802={x -2206.03101,y -1568.48901,z -46.4613991,a 40.3786583,b 1.76308298,c 3.98608398,s 2,t 11,e1 0.0,e2 0.0,e3 0.0,e4 0.0,e5 0.0,e6 0.0}
DECL FDAT Fp1802={TOOL_NO 1,BASE_NO 2,IPO_FRAME #BASE}
DECL PDAT PPDAT11={VEL 100.0,ACC 80.0,APO_DIST 50.0}
DECL E6POS XP1803={x -2382.18701,y -1952.18103,z -41.4048996,a 68.9136734,b 1.83556795,c 4.3166461,s 2,t 11,e1 0.0,e2 0.0,e3 0.0,e4 0.0,e5 0.0,e6 0.0}
DECL FDAT Fp1803={TOOL_NO 1,BASE_NO 2,IPO_FRAME #BASE}
DECL PDAT PPDAT12={VEL 100.0,ACC 80.0,APO_DIST 50.0}
DECL E6POS XP1804={x -2382.18701,y -1952.18103,z -41.4048996,a 68.9136734,b 1.83556795,c 4.3166461,s 2,t 11,e1 0.0,e2 0.0,e3 0.0,e4 0.0,e5 0.0,e6 0.0}
DECL FDAT Fp1804={TOOL_NO 1,BASE_NO 2,IPO_FRAME #BASE}
DECL PDAT PPDAT13={VEL 100.0,ACC 80.0,APO_DIST 50.0}
DECL E6POS XP1805={x -320.147797,y -2374.71606,z -105.432297,a -2.63908291,b -0.573716819,c 0.858778179,s 2,t 10,e1 0.0,e2 0.0,e3 0.0,e4 0.0,e5 0.0,e6 0.0}
DECL FDAT Fp1805={TOOL_NO 1,BASE_NO 2,IPO_FRAME #BASE}
DECL PDAT PPDAT14={VEL 100.0,ACC 80.0,APO_DIST 100.0}
DECL E6POS XP1806={x 216.575195,y -1858.94104,z 272.276215,a -84.0282669,b -3.96446896,c 12.2368097,s 2,t 10,e1 0.0,e2 0.0,e3 0.0,e4 0.0,e5 0.0,e6 0.0}
DECL FDAT Fp1806={TOOL_NO 1,BASE_NO 0,IPO_FRAME #BASE}
DECL PDAT PPDAT15={VEL 100.0,ACC 85.0,APO_DIST 100.0}
DECL E6POS XP1807={x -268.966095,y -1219.13098,z 454.964111,a -92.7284012,b -0.811235487,c 1.50273204,s 2,t 10,e1 0.0,e2 0.0,e3 0.0,e4 0.0,e5 0.0,e6 0.0}
DECL FDAT Fp1807={TOOL_NO 1,BASE_NO 0,IPO_FRAME #BASE}
DECL PDAT PPDAT16={VEL 100.0,ACC 85.0,APO_DIST 100.0}
DECL E6POS XP1808={x 1162.25403,y -212.311295,z 514.02887,a -114.784103,b 1.14916301,c 4.29522991,s 2,t 2,e1 0.0,e2 0.0,e3 0.0,e4 0.0,e5 0.0,e6 0.0}
DECL FDAT Fp1808={TOOL_NO 1,BASE_NO 0,IPO_FRAME #BASE}
DECL PDAT PPDAT17={VEL 100.0,ACC 85.0,APO_DIST 10.0}
DECL E6POS XP1809={x 1478.77502,y -1347.04602,z 884.754578,a -82.0556564,b -65.1650925,c 3.7185061,s 2,t 2,e1 0.0,e2 0.0,e3 0.0,e4 0.0,e5 0.0,e6 0.0}
DECL FDAT Fp1809={TOOL_NO 1,BASE_NO 0,IPO_FRAME #BASE}
DECL PDAT PPDAT18={VEL 100.0,ACC 85.0,APO_DIST 10.0}
DECL E6POS XP1810={x 1264.39905,y -1657.29297,z 945.626709,a -88.5366211,b -65.2689819,c -0.315103203,s 2,t 2,e1 0.0,e2 0.0,e3 0.0,e4 0.0,e5 0.0,e6 0.0}
DECL FDAT Fp1810={TOOL_NO 1,BASE_NO 0,IPO_FRAME #BASE}
DECL PDAT PPDAT19={VEL 100.0,ACC 85.0,APO_DIST 10.0}
DECL E6POS XP1811={x 1267.11597,y -1658.28796,z 1022.599,a -76.2749329,b -71.7416229,c -3.91462493,s 2,t 2,e1 0.0,e2 0.0,e3 0.0,e4 0.0,e5 0.0,e6 0.0}
DECL FDAT Fp1811={TOOL_NO 1,BASE_NO 0,IPO_FRAME #BASE}
DECL PDAT PPDAT20={VEL 100.0,ACC 85.0,APO_DIST 10.0}
DECL E6POS XP1812={x 1290.60803,y -1657.93103,z 963.055481,a -76.2796783,b -71.7437134,c -3.90588307,s 2,t 2,e1 0.0,e2 0.0,e3 0.0,e4 0.0,e5 0.0,e6 0.0}
DECL FDAT Fp1812={TOOL_NO 1,BASE_NO 0,IPO_FRAME #BASE}
DECL PDAT PPDAT21={VEL 100.0,ACC 85.0,APO_DIST 10.0}
DECL E6POS XP1813={x 1367.02295,y -1526.10095,z 859.774719,a -87.2438278,b -63.3831291,c 3.37517595,s 2,t 2,e1 0.0,e2 0.0,e3 0.0,e4 0.0,e5 0.0,e6 0.0}
DECL FDAT Fp1813={TOOL_NO 1,BASE_NO 0,IPO_FRAME #BASE}
DECL PDAT PPDAT22={VEL 100.0,ACC 85.0,APO_DIST 10.0}
DECL E6POS XP1814={x 1092.26404,y -417.520691,z 244.1436,a -96.5515366,b -8.95622635,c 4.26685381,s 2,t 2,e1 0.0,e2 0.0,e3 0.0,e4 0.0,e5 0.0,e6 0.0}
DECL FDAT Fp1814={TOOL_NO 1,BASE_NO 0,IPO_FRAME #BASE}
DECL PDAT PPDAT23={VEL 100.0,ACC 85.0,APO_DIST 10.0}
DECL E6POS XP1815={x 875.951172,y -127.552101,z 429.440887,a -90.4922104,b 0.331040293,c 3.53013206,s 2,t 10,e1 0.0,e2 0.0,e3 0.0,e4 0.0,e5 0.0,e6 0.0}
DECL FDAT Fp1815={TOOL_NO 1,BASE_NO 0,IPO_FRAME #BASE}
DECL PDAT PPDAT24={VEL 100.0,ACC 85.0,APO_DIST 10.0}
DECL E6POS XP1816={x 801.707825,y -406.20459,z 473.218109,a -115.815598,b 0.051684469,c 3.53548908,s 2,t 2,e1 0.0,e2 0.0,e3 0.0,e4 0.0,e5 0.0,e6 0.0}
DECL FDAT Fp1816={TOOL_NO 1,BASE_NO 0,IPO_FRAME #BASE}
DECL PDAT PPDAT25={VEL 100.0,ACC 85.0,APO_DIST 10.0}
DECL E6POS XP1817={x 688.968079,y -612.917175,z 384.596893,a -129.337296,b 0.0517537408,c 3.53589201,s 2,t 2,e1 0.0,e2 0.0,e3 0.0,e4 0.0,e5 0.0,e6 0.0}
DECL FDAT Fp1817={TOOL_NO 1,BASE_NO 0,IPO_FRAME #BASE}
DECL PDAT PPDAT26={VEL 100.0,ACC 85.0,APO_DIST 10.0}
DECL E6POS XP1818={x 401.636993,y -721.835327,z 414.848999,a -153.425995,b 0.0325570405,c 0.645587087,s 2,t 2,e1 0.0,e2 0.0,e3 0.0,e4 0.0,e5 0.0,e6 0.0}
DECL FDAT Fp1818={TOOL_NO 1,BASE_NO 0,IPO_FRAME #BASE}
DECL PDAT PPDAT27={VEL 100.0,ACC 85.0,APO_DIST 10.0}
DECL E6POS XSWP_60_0005={x 1267.11597,y -1658.28796,z 1022.599,a -76.2749329,b -71.7416229,c -3.91462493,s 2,t 2,e1 0.0,e2 0.0,e3 0.0,e4 0.0,e5 0.0,e6 0.0}
DECL FDAT FSWP_60_0005={TOOL_NO 1,BASE_NO 0,IPO_FRAME #BASE}
DECL E6POS XSWP_62_0005={x 1267.15601,y -1658.25903,z 1024.21594,a -76.2778778,b -71.7415085,c -3.91174507,s 2,t 2,e1 0.0,e2 0.0,e3 0.0,e4 0.0,e5 0.0,e6 0.0}
DECL FDAT FSWP_62_0005={TOOL_NO 1,BASE_NO 0,IPO_FRAME #BASE}
DECL E6POS XP1819={x 1294.42896,y -1086.45605,z 593.15271,a -90.0058594,b -38.7629509,c 7.58146286,s 2,t 2,e1 0.0,e2 0.0,e3 0.0,e4 0.0,e5 0.0,e6 0.0}
DECL FDAT Fp1819={TOOL_NO 1,BASE_NO 0,IPO_FRAME #BASE}
DECL PDAT PPDAT28={VEL 100.0,ACC 85.0,APO_DIST 10.0}
DECL E6POS XP1820={x 1351.16602,y -1521.03296,z 1310.87402,a -165.300507,b 2.66181707,c 71.3331299,s 2,t 34,e1 0.0,e2 0.0,e3 0.0,e4 0.0,e5 0.0,e6 0.0}
DECL FDAT Fp1820={TOOL_NO 1,BASE_NO 0,IPO_FRAME #BASE}
DECL PDAT PPDAT29={VEL 100.0,ACC 85.0,APO_DIST 10.0}
DECL E6POS XP1821={x 1350.67004,y -1866.52698,z 1365.66895,a -156.353897,b -5.2249651,c 61.3996887,s 2,t 34,e1 0.0,e2 0.0,e3 0.0,e4 0.0,e5 0.0,e6 0.0}
DECL FDAT Fp1821={TOOL_NO 1,BASE_NO 0,IPO_FRAME #BASE}
DECL PDAT PPDAT30={VEL 100.0,ACC 85.0,APO_DIST 10.0}
DECL E6POS XP1822={x 1215.552,y -1863.63501,z 1366.95703,a -156.353806,b -5.22543812,c 61.3993683,s 2,t 34,e1 0.0,e2 0.0,e3 0.0,e4 0.0,e5 0.0,e6 0.0}
DECL FDAT Fp1822={TOOL_NO 1,BASE_NO 0,IPO_FRAME #BASE}
DECL PDAT PPDAT31={VEL 100.0,ACC 85.0,APO_DIST 10.0}
DECL E6POS XP1823={x 1200.84998,y -1856.62402,z 1370.56494,a -156.356003,b -5.17883587,c 61.4194298,s 2,t 34,e1 0.0,e2 0.0,e3 0.0,e4 0.0,e5 0.0,e6 0.0}
DECL FDAT Fp1823={TOOL_NO 1,BASE_NO 0,IPO_FRAME #BASE}
DECL PDAT PPDAT32={VEL 100.0,ACC 85.0,APO_DIST 10.0}
DECL E6POS XP1824={x 319.441803,y -892.141113,z 790.858215,a -66.2261581,b -5.64948797,c 60.9168701,s 2,t 34,e1 0.0,e2 0.0,e3 0.0,e4 0.0,e5 0.0,e6 0.0}
DECL FDAT Fp1824={TOOL_NO 1,BASE_NO 2,IPO_FRAME #BASE}
DECL PDAT PPDAT33={VEL 50.0,ACC 100.0,APO_DIST 10.0}
DECL E6POS XP1825={x 1208.94604,y -1867.84595,z 1366.96399,a -156.353897,b -5.22473717,c 61.3997002,s 2,t 34,e1 0.0,e2 0.0,e3 0.0,e4 0.0,e5 0.0,e6 0.0}
DECL FDAT Fp1825={TOOL_NO 1,BASE_NO 0,IPO_FRAME #BASE}
DECL PDAT PPDAT34={VEL 100.0,ACC 85.0,APO_DIST 10.0}
DECL E6POS XP1826={x 1272.81494,y -1880.90796,z 1407.51501,a -156.355194,b -5.22684002,c 61.3990211,s 2,t 34,e1 0.0,e2 0.0,e3 0.0,e4 0.0,e5 0.0,e6 0.0}
DECL FDAT Fp1826={TOOL_NO 1,BASE_NO 0,IPO_FRAME #BASE}
DECL PDAT PPDAT35={VEL 100.0,ACC 85.0,APO_DIST 10.0}
DECL E6POS XP1827={x 1279.70703,y -1895.32898,z 1473.25195,a -156.352005,b -5.22255182,c 61.4003906,s 2,t 34,e1 0.0,e2 0.0,e3 0.0,e4 0.0,e5 0.0,e6 0.0}
DECL FDAT Fp1827={TOOL_NO 1,BASE_NO 0,IPO_FRAME #BASE}
DECL PDAT PPDAT36={VEL 100.0,ACC 85.0,APO_DIST 10.0}
DECL E6POS XP1828={x 1220.31995,y -1918.66296,z 1469.62097,a -156.354706,b -5.22167587,c 61.3990707,s 2,t 2,e1 0.0,e2 0.0,e3 0.0,e4 0.0,e5 0.0,e6 0.0}
DECL FDAT Fp1828={TOOL_NO 1,BASE_NO 0,IPO_FRAME #BASE}
DECL PDAT PPDAT37={VEL 100.0,ACC 85.0,APO_DIST 10.0}
DECL E6POS XP1829={x 373.9758,y -880.796814,z 896.996521,a -66.2239685,b -5.69177818,c 60.8968315,s 2,t 2,e1 0.0,e2 0.0,e3 0.0,e4 0.0,e5 0.0,e6 0.0}
DECL FDAT Fp1829={TOOL_NO 1,BASE_NO 2,IPO_FRAME #BASE}
DECL PDAT PPDAT38={VEL 50.0,ACC 100.0,APO_DIST 10.0}
DECL E6POS XP1830={x 1220.31995,y -1918.66394,z 1469.61597,a -156.354797,b -5.22175789,c 61.3990097,s 2,t 2,e1 0.0,e2 0.0,e3 0.0,e4 0.0,e5 0.0,e6 0.0}
DECL FDAT Fp1830={TOOL_NO 1,BASE_NO 0,IPO_FRAME #BASE}
DECL PDAT PPDAT39={VEL 100.0,ACC 85.0,APO_DIST 10.0}
DECL E6POS XP1831={x 1279.70605,y -1895.33997,z 1473.20898,a -156.352402,b -5.22327185,c 61.3990402,s 2,t 34,e1 0.0,e2 0.0,e3 0.0,e4 0.0,e5 0.0,e6 0.0}
DECL FDAT Fp1831={TOOL_NO 1,BASE_NO 0,IPO_FRAME #BASE}
DECL PDAT PPDAT40={VEL 100.0,ACC 85.0,APO_DIST 10.0}
DECL E6POS XP1832={x 1351.172,y -1521.03503,z 1310.89294,a -165.300293,b 2.66227603,c 71.3338776,s 2,t 34,e1 0.0,e2 0.0,e3 0.0,e4 0.0,e5 0.0,e6 0.0}
DECL FDAT Fp1832={TOOL_NO 1,BASE_NO 0,IPO_FRAME #BASE}
DECL PDAT PPDAT41={VEL 100.0,ACC 85.0,APO_DIST 10.0}
DECL E6POS XP1833={x 1367.026,y -1526.10999,z 859.788208,a -87.2437668,b -63.3836288,c 3.37530994,s 2,t 2,e1 0.0,e2 0.0,e3 0.0,e4 0.0,e5 0.0,e6 0.0}
DECL FDAT Fp1833={TOOL_NO 1,BASE_NO 0,IPO_FRAME #BASE}
DECL PDAT PPDAT42={VEL 100.0,ACC 85.0,APO_DIST 10.0}
DECL E6POS XP1834={x -3701.63696,y -2031.15295,z 1324.87402,a 86.1747437,b 15.1261702,c 74.728447,s 2,t 3,e1 0.0,e2 0.0,e3 0.0,e4 0.0,e5 0.0,e6 0.0}
DECL FDAT Fp1834={TOOL_NO 1,BASE_NO 2,IPO_FRAME #BASE}
DECL PDAT PPDAT43={VEL 100.0,ACC 80.0,APO_DIST 10.0}
ENDDAT
